  [776] = {x=-522, y=87.731, z=176, rx=180, rz=-85.738, shoulder=lefty, elbow=epositive, wrist=wpositive, fatherId=fReference[0]}
  [777] = {x=-519.753, y=117.878, z=176, rx=180, rz=-72.47, shoulder=lefty, elbow=epositive, wrist=wpositive, fatherId=fReference[0]}
  [778] = {x=-510.651, y=146.693, z=176, rx=180, rz=-58.912, shoulder=lefty, elbow=epositive, wrist=wpositive, fatherId=fReference[0]}
  [779] = {x=-495.048, y=172.571, z=176, rx=180, rz=-45.354, shoulder=lefty, elbow=epositive, wrist=wpositive, fatherId=fReference[0]}
  [780] = {x=-473.813, y=194.069, z=176, rx=180, rz=-31.796, shoulder=lefty, elbow=epositive, wrist=wpositive, fatherId=fReference[0]}
  [781] = {x=-448.13, y=209.991, z=176, rx=180, rz=-18.238, shoulder=lefty, elbow=epositive, wrist=wpositive, fatherId=fReference[0]}
  [782] = {x=-419.43, y=219.448, z=176, rx=180, rz=-4.843, shoulder=lefty, elbow=epositive, wrist=wpositive, fatherId=fReference[0]}
  [783] = {x=-389.312, y=222, z=176, rx=180, shoulder=lefty, elbow=epositive, wrist=wpositive, fatherId=fReference[0]}
  [784] = {x=-359.024, y=222, z=176, rx=180, shoulder=lefty, elbow=epositive, wrist=wpositive, fatherId=fReference[0]}
  [785] = {x=-328.735, y=222, z=176, rx=-180, shoulder=lefty, elbow=epositive, wrist=wpositive, fatherId=fReference[0]}
  [786] = {x=-298.447, y=222, z=176, rx=180, shoulder=lefty, elbow=epositive, wrist=wpositive, fatherId=fReference[0]}
  [787] = {x=-268.159, y=222, z=176, rx=180, shoulder=lefty, elbow=epositive, wrist=wpositive, fatherId=fReference[0]}
  [788] = {x=-237.87, y=222, z=176, rx=-180, shoulder=lefty, elbow=epositive, wrist=wpositive, fatherId=fReference[0]}
  [789] = {x=-207.582, y=222, z=176, rx=180, shoulder=lefty, elbow=epositive, wrist=wpositive, fatherId=fReference[0]}
  [790] = {x=-177.293, y=222, z=176, rx=180, shoulder=lefty, elbow=epositive, wrist=wpositive, fatherId=fReference[0]}
  [791] = {x=-147.005, y=222, z=176, rx=-180, shoulder=lefty, elbow=epositive, wrist=wpositive, fatherId=fReference[0]}
  [792] = {x=-116.716, y=222, z=176, rx=180, shoulder=lefty, elbow=epositive, wrist=wpositive, fatherId=fReference[0]}
  [793] = {x=-86.428, y=222, z=176, rx=180, shoulder=lefty, elbow=epositive, wrist=wpositive, fatherId=fReference[0]}
  [794] = {x=-56.139, y=222, z=176, rx=180, shoulder=lefty, elbow=epositive, wrist=wpositive, fatherId=fReference[0]}
  [795] = {x=-25.851, y=222, z=176, rx=-180, shoulder=lefty, elbow=epositive, wrist=wpositive, fatherId=fReference[0]}
  [796] = {x=4.437, y=222, z=176, rx=-180, shoulder=lefty, elbow=epositive, wrist=wpositive, fatherId=fReference[0]}
  [797] = {x=34.726, y=222, z=176, rx=-180, shoulder=lefty, elbow=epositive, wrist=wpositive, fatherId=fReference[0]}
  [798] = {x=65.014, y=222, z=176, rx=180, shoulder=lefty, elbow=epositive, wrist=wpositive, fatherId=fReference[0]}
  [799] = {x=95.303, y=222, z=176, rx=180, shoulder=lefty, elbow=epositive, wrist=wpositive, fatherId=fReference[0]}
  [800] = {x=125.591, y=222, z=176, rx=-180, shoulder=lefty, elbow=epositive, wrist=wpositive, fatherId=fReference[0]}
  [801] = {x=155.88, y=222, z=176, rx=180, shoulder=lefty, elbow=epositive, wrist=wpositive, fatherId=fReference[0]}
  [802] = {x=186.168, y=222, z=176, rx=180, shoulder=lefty, elbow=epositive, wrist=wpositive, fatherId=fReference[0]}
  [803] = {x=216.456, y=222, z=176, rx=180, shoulder=lefty, elbow=epositive, wrist=wpositive, fatherId=fReference[0]}
  [804] = {x=246.745, y=222, z=176, rx=180, shoulder=lefty, elbow=epositive, wrist=wpositive, fatherId=fReference[0]}
  [805] = {x=277.033, y=222, z=176, rx=180, shoulder=lefty, elbow=epositive, wrist=wpositive, fatherId=fReference[0]}
  [806] = {x=307.322, y=222, z=176, rx=-180, shoulder=lefty, elbow=epositive, wrist=wpositive, fatherId=fReference[0]}
  [807] = {x=337.61, y=222, z=176, rx=180, shoulder=lefty, elbow=epositive, wrist=wpositive, fatherId=fReference[0]}
  [808] = {x=367.899, y=222, z=176, rx=-180, rz=0.13, shoulder=lefty, elbow=epositive, wrist=wpositive, fatherId=fReference[0]}
  [809] = {x=398.186, y=221.932, z=176, rx=180, rz=8.653, shoulder=lefty, elbow=epositive, wrist=wpositive, fatherId=fReference[0]}
  [810] = {x=428.06, y=217.385, z=176, rx=180, rz=22.211, shoulder=lefty, elbow=epositive, wrist=wpositive, fatherId=fReference[0]}
  [811] = {x=456.036, y=205.962, z=176, rx=-180, rz=35.769, shoulder=lefty, elbow=epositive, wrist=wpositive, fatherId=fReference[0]}
  [812] = {x=480.554, y=188.3, z=176, rx=-180, rz=49.327, shoulder=lefty, elbow=epositive, wrist=wpositive, fatherId=fReference[0]}
  [813] = {x=500.248, y=165.381, z=176, rx=180, rz=62.884, shoulder=lefty, elbow=epositive, wrist=wpositive, fatherId=fReference[0]}
  [814] = {x=514.021, y=138.485, z=176, rx=-180, rz=76.442, shoulder=lefty, elbow=epositive, wrist=wpositive, fatherId=fReference[0]}
  [815] = {x=521.105, y=109.109, z=176, rx=-180, rz=88.306, shoulder=lefty, elbow=epositive, wrist=wpositive, fatherId=fReference[0]}
  [816] = {x=522, y=78.856, z=176, rx=180, rz=90, shoulder=lefty, elbow=epositive, wrist=wpositive, fatherId=fReference[0]}
  [817] = {x=522, y=48.567, z=176, rx=180, rz=90, shoulder=lefty, elbow=epositive, wrist=wpositive, fatherId=fReference[0]}
  [818] = {x=522, y=18.279, z=176, rx=180, rz=90, shoulder=lefty, elbow=epositive, wrist=wpositive, fatherId=fReference[0]}
  [819] = {x=522, y=-12.01, z=176, rx=180, rz=90, shoulder=lefty, elbow=epositive, wrist=wpositive, fatherId=fReference[0]}
  [820] = {x=522, y=-42.298, z=176, rx=180, rz=90, shoulder=lefty, elbow=epositive, wrist=wpositive, fatherId=fReference[0]}
  [821] = {x=522, y=-72.586, z=176, rx=180, rz=90.582, shoulder=lefty, elbow=epositive, wrist=wpositive, fatherId=fReference[0]}
  [822] = {x=521.692, y=-102.868, z=176, rx=180, rz=100.751, shoulder=lefty, elbow=epositive, wrist=wpositive, fatherId=fReference[0]}
  [823] = {x=516.055, y=-132.555, z=176, rx=180, rz=114.309, shoulder=lefty, elbow=epositive, wrist=wpositive, fatherId=fReference[0]}
  [824] = {x=503.616, y=-160.094, z=176, rx=180, rz=127.867, shoulder=lefty, elbow=epositive, wrist=wpositive, fatherId=fReference[0]}
  [825] = {x=485.067, y=-183.949, z=176, rx=180, rz=141.425, shoulder=lefty, elbow=epositive, wrist=wpositive, fatherId=fReference[0]}
  [826] = {x=461.443, y=-202.791, z=176, rx=180, rz=154.983, shoulder=lefty, elbow=epositive, wrist=wpositive, fatherId=fReference[0]}
  [827] = {x=434.06, y=-215.57, z=176, rx=-180, rz=168.541, shoulder=lefty, elbow=epositive, wrist=wpositive, fatherId=fReference[0]}
  [828] = {x=404.445, y=-221.573, z=176, rx=-180, rz=176.192, shoulder=lefty, elbow=epositive, wrist=wpositive, fatherId=fReference[0]}
  [829] = {x=374.168, y=-222, z=176, rx=-180, rz=177, shoulder=lefty, elbow=epositive, wrist=wpositive, fatherId=fReference[0]}
  [830] = {x=343.88, y=-222, z=176, rx=-180, rz=178, shoulder=lefty, elbow=epositive, wrist=wpositive, fatherId=fReference[0]}
  [831] = {x=313.591, y=-222, z=176, rx=-180, rz=179, shoulder=lefty, elbow=epositive, wrist=wpositive, fatherId=fReference[0]}
  [832] = {x=283.303, y=-222, z=176, rx=180, rz=-180, shoulder=lefty, elbow=epositive, wrist=wpositive, fatherId=fReference[0]}
  [833] = {x=253.014, y=-222, z=176, rx=180, rz=-180, shoulder=lefty, elbow=epositive, wrist=wpositive, fatherId=fReference[0]}
  [834] = {x=222.726, y=-222, z=176, rx=-180, rz=-180, shoulder=lefty, elbow=epositive, wrist=wpositive, fatherId=fReference[0]}
  [835] = {x=192.437, y=-222, z=176, rx=-180, rz=-180, shoulder=lefty, elbow=epositive, wrist=wpositive, fatherId=fReference[0]}
  [836] = {x=162.149, y=-222, z=176, rx=180, rz=-180, shoulder=lefty, elbow=epositive, wrist=wpositive, fatherId=fReference[0]}
  [837] = {x=131.861, y=-222, z=176, rx=-180, rz=-180, shoulder=lefty, elbow=epositive, wrist=wpositive, fatherId=fReference[0]}
  [838] = {x=101.572, y=-222, z=176, rx=180, rz=-180, shoulder=lefty, elbow=epositive, wrist=wpositive, fatherId=fReference[0]}
  [839] = {x=71.284, y=-222, z=176, rx=-180, rz=-180, shoulder=lefty, elbow=epositive, wrist=wpositive, fatherId=fReference[0]}
  [840] = {x=40.995, y=-222, z=176, rx=180, rz=-180, shoulder=lefty, elbow=epositive, wrist=wpositive, fatherId=fReference[0]}
  [841] = {x=10.707, y=-222, z=176, rx=180, rz=-180, shoulder=lefty, elbow=epositive, wrist=wpositive, fatherId=fReference[0]}
  [842] = {x=-19.582, y=-222, z=176, rx=180, rz=-180, shoulder=lefty, elbow=epositive, wrist=wpositive, fatherId=fReference[0]}
  [843] = {x=-49.87, y=-222, z=176, rx=-180, rz=-180, shoulder=lefty, elbow=epositive, wrist=wpositive, fatherId=fReference[0]}
  [844] = {x=-80.159, y=-222, z=176, rx=-180, rz=-180, shoulder=lefty, elbow=epositive, wrist=wpositive, fatherId=fReference[0]}
  [845] = {x=-110.447, y=-222, z=176, rx=180, rz=-180, shoulder=lefty, elbow=epositive, wrist=wpositive, fatherId=fReference[0]}
  [846] = {x=-140.735, y=-222, z=176, rx=180, rz=-180, shoulder=lefty, elbow=epositive, wrist=wpositive, fatherId=fReference[0]}
  [847] = {x=-171.024, y=-222, z=176, rx=180, rz=-180, shoulder=lefty, elbow=epositive, wrist=wpositive, fatherId=fReference[0]}
  [848] = {x=-201.312, y=-222, z=176, rx=180, rz=-180, shoulder=lefty, elbow=epositive, wrist=wpositive, fatherId=fReference[0]}
  [849] = {x=-231.601, y=-222, z=176, rx=180, rz=-180, shoulder=lefty, elbow=epositive, wrist=wpositive, fatherId=fReference[0]}
  [850] = {x=-261.889, y=-222, z=176, rx=-180, rz=-180, shoulder=lefty, elbow=epositive, wrist=wpositive, fatherId=fReference[0]}
  [851] = {x=-292.178, y=-222, z=176, rx=180, rz=-180, shoulder=lefty, elbow=epositive, wrist=wpositive, fatherId=fReference[0]}
  [852] = {x=-322.466, y=-222, z=176, rx=180, rz=-180, shoulder=lefty, elbow=epositive, wrist=wpositive, fatherId=fReference[0]}
  [853] = {x=-352.754, y=-222, z=176, rx=-180, rz=-180, shoulder=lefty, elbow=epositive, wrist=wpositive, fatherId=fReference[0]}
  [854] = {x=-383.043, y=-222, z=176, rx=-180, rz=-177.239, shoulder=lefty, elbow=epositive, wrist=wpositive, fatherId=fReference[0]}
  [855] = {x=-413.258, y=-220.543, z=176, rx=180, rz=-164.568, shoulder=lefty, elbow=epositive, wrist=wpositive, fatherId=fReference[0]}
  [856] = {x=-442.386, y=-212.502, z=176, rx=180, rz=-157.01, shoulder=lefty, elbow=epositive, wrist=wpositive, fatherId=fReference[0]}
  [857] = {x=-468.818, y=-197.857, z=176, rx=-180, rz=-156.452, shoulder=lefty, elbow=epositive, wrist=wpositive, fatherId=fReference[0]}
  [858] = {x=-491.08, y=-177.424, z=176, rx=180, rz=-154.895, shoulder=lefty, elbow=epositive, wrist=wpositive, fatherId=fReference[0]}
  [859] = {x=-507.931, y=-152.341, z=176, rx=-180, rz=-154.337, shoulder=lefty, elbow=epositive, wrist=wpositive, fatherId=fReference[0]}
  [860] = {x=-518.433, y=-124.007, z=176, rx=180, rz=-153.779, shoulder=lefty, elbow=epositive, wrist=wpositive, fatherId=fReference[0]}
  [861] = {x=-522, y=-94, z=176, rx=180, rz=-152.779, shoulder=lefty, elbow=epositive, wrist=wpositive, fatherId=fReference[0]}
  [862] = {x=-522, y=-94, z=176, rx=180, rz=-152.779, shoulder=lefty, elbow=epositive, wrist=wpositive, fatherId=fReference[0]}
  [863] = {x=-522, y=-94, z=276, rx=-180, rz=-152.779, shoulder=lefty, elbow=epositive, wrist=wpositive, fatherId=fReference[0]}
  [864] = {x=-477.591, y=-88.721, z=287.443, rx=176.622, ry=-26.365, rz=160.43, shoulder=lefty, elbow=epositive, wrist=wpositive, fatherId=fReference[0]}
  [865] = {x=-522, y=-94, z=198, rx=176.622, ry=-26.365, rz=-18.57, shoulder=lefty, elbow=epositive, wrist=wpositive, fatherId=fReference[0]}
  [866] = {x=-522, y=-94, z=198, rx=176.622, ry=-26.365, rz=-97.57, shoulder=lefty, elbow=epositive, wrist=wpositive, fatherId=fReference[0]}
  [867] = {x=-518.433, y=-124.007, z=198, rx=176.622, ry=-26.365, rz=-109.742, shoulder=lefty, elbow=epositive, wrist=wpositive, fatherId=fReference[0]}
  [868] = {x=-507.931, y=-152.341, z=198, rx=170.142, ry=-24.793, rz=-124.68, shoulder=lefty, elbow=epositive, wrist=wpositive, fatherId=fReference[0]}
  [869] = {x=-491.08, y=-177.424, z=198, rx=164.42, ry=-21.791, rz=-139.083, shoulder=lefty, elbow=epositive, wrist=wpositive, fatherId=fReference[0]}
  [870] = {x=-468.818, y=-197.857, z=198, rx=159.778, ry=-17.602, rz=-152.787, shoulder=lefty, elbow=epositive, wrist=wpositive, fatherId=fReference[0]}
  [871] = {x=-442.386, y=-212.502, z=198, rx=156.378, ry=-12.518, rz=-165.809, shoulder=lefty, elbow=epositive, wrist=wpositive, fatherId=fReference[0]}
  [872] = {x=-413.258, y=-220.543, z=198, rx=154.267, ry=-6.834, rz=-177.501, shoulder=lefty, elbow=epositive, wrist=wpositive, fatherId=fReference[0]}
  [873] = {x=-383.043, y=-222, z=198, rx=153.462, ry=-1.234, rz=-180, shoulder=lefty, elbow=epositive, wrist=wpositive, fatherId=fReference[0]}
  [874] = {x=-352.754, y=-222, z=198, rx=153.435, rz=-180, shoulder=lefty, elbow=epositive, wrist=wpositive, fatherId=fReference[0]}
  [875] = {x=-322.466, y=-222, z=198, rx=153.435, rz=-180, shoulder=lefty, elbow=epositive, wrist=wpositive, fatherId=fReference[0]}
  [876] = {x=-292.178, y=-222, z=198, rx=153.435, rz=-180, shoulder=lefty, elbow=epositive, wrist=wpositive, fatherId=fReference[0]}
  [877] = {x=-261.889, y=-222, z=198, rx=153.435, rz=-180, shoulder=lefty, elbow=epositive, wrist=wpositive, fatherId=fReference[0]}
  [878] = {x=-231.601, y=-222, z=198, rx=153.435, rz=-180, shoulder=lefty, elbow=epositive, wrist=wpositive, fatherId=fReference[0]}
  [879] = {x=-201.312, y=-222, z=198, rx=153.435, rz=-180, shoulder=lefty, elbow=epositive, wrist=wpositive, fatherId=fReference[0]}
  [880] = {x=-171.024, y=-222, z=198, rx=153.435, rz=-180, shoulder=lefty, elbow=epositive, wrist=wpositive, fatherId=fReference[0]}
  [881] = {x=-140.735, y=-222, z=198, rx=153.435, rz=-180, shoulder=lefty, elbow=epositive, wrist=wpositive, fatherId=fReference[0]}
  [882] = {x=-110.447, y=-222, z=198, rx=153.435, rz=-180, shoulder=lefty, elbow=epositive, wrist=wpositive, fatherId=fReference[0]}
  [883] = {x=-80.159, y=-222, z=198, rx=153.435, rz=-180, shoulder=lefty, elbow=epositive, wrist=wpositive, fatherId=fReference[0]}
  [884] = {x=-49.87, y=-222, z=198, rx=153.435, rz=-180, shoulder=lefty, elbow=epositive, wrist=wpositive, fatherId=fReference[0]}
  [885] = {x=-19.582, y=-222, z=198, rx=153.435, rz=-180, shoulder=lefty, elbow=epositive, wrist=wpositive, fatherId=fReference[0]}
  [886] = {x=10.707, y=-222, z=198, rx=153.435, rz=-180, shoulder=lefty, elbow=epositive, wrist=wpositive, fatherId=fReference[0]}
  [887] = {x=40.995, y=-222, z=198, rx=153.435, rz=-180, shoulder=lefty, elbow=epositive, wrist=wpositive, fatherId=fReference[0]}
  [888] = {x=71.284, y=-222, z=198, rx=153.435, rz=-180, shoulder=lefty, elbow=epositive, wrist=wpositive, fatherId=fReference[0]}
  [889] = {x=101.572, y=-222, z=198, rx=153.435, rz=-180, shoulder=lefty, elbow=epositive, wrist=wpositive, fatherId=fReference[0]}
  [890] = {x=131.861, y=-222, z=198, rx=153.435, rz=-180, shoulder=lefty, elbow=epositive, wrist=wpositive, fatherId=fReference[0]}
  [891] = {x=162.149, y=-222, z=198, rx=153.435, rz=-180, shoulder=lefty, elbow=epositive, wrist=wpositive, fatherId=fReference[0]}
  [892] = {x=192.437, y=-222, z=198, rx=153.435, rz=-180, shoulder=lefty, elbow=epositive, wrist=wpositive, fatherId=fReference[0]}
  [893] = {x=222.726, y=-222, z=198, rx=153.435, rz=-180, shoulder=lefty, elbow=epositive, wrist=wpositive, fatherId=fReference[0]}
  [894] = {x=253.014, y=-222, z=198, rx=153.435, rz=-180, shoulder=lefty, elbow=epositive, wrist=wpositive, fatherId=fReference[0]}
  [895] = {x=283.303, y=-222, z=198, rx=153.435, rz=-180, shoulder=lefty, elbow=epositive, wrist=wpositive, fatherId=fReference[0]}
  [896] = {x=313.591, y=-222, z=198, rx=153.435, rz=-175, shoulder=lefty, elbow=epositive, wrist=wpositive, fatherId=fReference[0]}
  [897] = {x=343.88, y=-222, z=198, rx=153.435, rz=-166, shoulder=lefty, elbow=epositive, wrist=wpositive, fatherId=fReference[0]}
  [898] = {x=374.168, y=-222, z=198, rx=153.435, rz=-157.722, shoulder=lefty, elbow=epositive, wrist=wpositive, fatherId=fReference[0]}
  [899] = {x=404.445, y=-221.573, z=198, rx=153.437, ry=0.361, rz=-156.272, shoulder=lefty, elbow=epositive, wrist=wpositive, fatherId=fReference[0]}
  [900] = {x=434.06, y=-215.57, z=198, rx=153.894, ry=5.097, rz=157.552, shoulder=lefty, elbow=epositive, wrist=wpositive, fatherId=fReference[0]}
  [901] = {x=461.443, y=-202.791, z=198, rx=155.625, ry=10.902, rz=145.173, shoulder=lefty, elbow=epositive, wrist=wpositive, fatherId=fReference[0]}
  [902] = {x=485.067, y=-183.949, z=198, rx=158.65, ry=16.192, rz=132.325, shoulder=lefty, elbow=epositive, wrist=wpositive, fatherId=fReference[0]}
  [903] = {x=503.616, y=-160.094, z=198, rx=162.938, ry=20.674, rz=118.83, shoulder=lefty, elbow=epositive, wrist=wpositive, fatherId=fReference[0]}
  [904] = {x=516.055, y=-132.555, z=198, rx=168.369, ry=24.052, rz=104.624, shoulder=lefty, elbow=epositive, wrist=wpositive, fatherId=fReference[0]}
  [905] = {x=521.692, y=-102.868, z=198, rx=174.671, ry=26.063, rz=92.871, shoulder=lefty, elbow=epositive, wrist=wpositive, fatherId=fReference[0]}
  [906] = {x=522, y=-72.586, z=198, rx=179.709, ry=26.564, rz=90.13, shoulder=lefty, elbow=epositive, wrist=wpositive, fatherId=fReference[0]}
  [907] = {x=522, y=-42.298, z=198, rx=180, ry=26.565, rz=90, shoulder=lefty, elbow=epositive, wrist=wpositive, fatherId=fReference[0]}
  [908] = {x=522, y=-12.01, z=198, rx=180, ry=26.565, rz=90, shoulder=lefty, elbow=epositive, wrist=wpositive, fatherId=fReference[0]}
  [909] = {x=522, y=18.279, z=198, rx=180, ry=26.565, rz=90, shoulder=lefty, elbow=epositive, wrist=wpositive, fatherId=fReference[0]}
  [910] = {x=522, y=48.567, z=198, rx=180, ry=26.565, rz=90, shoulder=lefty, elbow=epositive, wrist=wpositive, fatherId=fReference[0]}
  [911] = {x=522, y=78.856, z=198, rx=-180, ry=26.565, rz=88.485, shoulder=lefty, elbow=epositive, wrist=wpositive, fatherId=fReference[0]}
  [912] = {x=521.105, y=109.109, z=198, rx=-179.153, ry=26.553, rz=77.465, shoulder=lefty, elbow=epositive, wrist=wpositive, fatherId=fReference[0]}
  [913] = {x=514.021, y=138.485, z=198, rx=-173.315, ry=25.769, rz=62.74, shoulder=lefty, elbow=epositive, wrist=wpositive, fatherId=fReference[0]}
  [914] = {x=500.248, y=165.381, z=198, rx=-167.162, ry=23.457, rz=48.037, shoulder=lefty, elbow=epositive, wrist=wpositive, fatherId=fReference[0]}
  [915] = {x=480.554, y=188.3, z=198, rx=-161.951, ry=19.827, rz=33.975, shoulder=lefty, elbow=epositive, wrist=wpositive, fatherId=fReference[0]}
  [916] = {x=456.036, y=205.962, z=198, rx=-157.918, ry=15.153, rz=20.624, shoulder=lefty, elbow=epositive, wrist=wpositive, fatherId=fReference[0]}
  [917] = {x=428.06, y=217.385, z=198, rx=-155.161, ry=9.733, rz=7.891, shoulder=lefty, elbow=epositive, wrist=wpositive, fatherId=fReference[0]}
  [918] = {x=398.186, y=221.932, z=198, rx=-153.696, ry=3.858, rz=1.116, shoulder=lefty, elbow=epositive, wrist=wpositive, fatherId=fReference[0]}
  [919] = {x=367.899, y=222, z=198, rx=-153.435, ry=0.058, shoulder=lefty, elbow=epositive, wrist=wpositive, fatherId=fReference[0]}
  [920] = {x=337.61, y=222, z=198, rx=-153.435, shoulder=lefty, elbow=epositive, wrist=wpositive, fatherId=fReference[0]}
  [921] = {x=307.322, y=222, z=198, rx=-153.435, shoulder=lefty, elbow=epositive, wrist=wpositive, fatherId=fReference[0]}
  [922] = {x=277.033, y=222, z=198, rx=-153.435, rz=1, shoulder=lefty, elbow=epositive, wrist=wpositive, fatherId=fReference[0]}
  [923] = {x=246.745, y=222, z=198, rx=-153.435, rz=2, shoulder=lefty, elbow=epositive, wrist=wpositive, fatherId=fReference[0]}
  [924] = {x=216.456, y=222, z=198, rx=-153.435, rz=2, shoulder=lefty, elbow=epositive, wrist=wpositive, fatherId=fReference[0]}
  [925] = {x=186.168, y=222, z=198, rx=-153.435, rz=3, shoulder=lefty, elbow=epositive, wrist=wpositive, fatherId=fReference[0]}
  [926] = {x=155.88, y=222, z=198, rx=-153.435, rz=4, shoulder=lefty, elbow=epositive, wrist=wpositive, fatherId=fReference[0]}
  [927] = {x=125.591, y=222, z=198, rx=-153.435, rz=4, shoulder=lefty, elbow=epositive, wrist=wpositive, fatherId=fReference[0]}
  [928] = {x=95.303, y=222, z=198, rx=-153.435, rz=5, shoulder=lefty, elbow=epositive, wrist=wpositive, fatherId=fReference[0]}
  [929] = {x=65.014, y=222, z=198, rx=-153.435, rz=6, shoulder=lefty, elbow=epositive, wrist=wpositive, fatherId=fReference[0]}
  [930] = {x=34.726, y=222, z=198, rx=-153.435, rz=7, shoulder=lefty, elbow=epositive, wrist=wpositive, fatherId=fReference[0]}
  [931] = {x=4.437, y=222, z=198, rx=-153.435, rz=7, shoulder=lefty, elbow=epositive, wrist=wpositive, fatherId=fReference[0]}
  [932] = {x=-25.851, y=222, z=198, rx=-153.435, rz=8, shoulder=lefty, elbow=epositive, wrist=wpositive, fatherId=fReference[0]}
  [933] = {x=-56.139, y=222, z=198, rx=-153.435, rz=9, shoulder=lefty, elbow=epositive, wrist=wpositive, fatherId=fReference[0]}
  [934] = {x=-86.428, y=222, z=198, rx=-153.435, rz=10, shoulder=lefty, elbow=epositive, wrist=wpositive, fatherId=fReference[0]}
  [935] = {x=-116.716, y=222, z=198, rx=-153.435, rz=10, shoulder=lefty, elbow=epositive, wrist=wpositive, fatherId=fReference[0]}
  [936] = {x=-147.005, y=222, z=198, rx=-153.435, rz=11, shoulder=lefty, elbow=epositive, wrist=wpositive, fatherId=fReference[0]}
  [937] = {x=-177.293, y=222, z=198, rx=-153.435, rz=12, shoulder=lefty, elbow=epositive, wrist=wpositive, fatherId=fReference[0]}
  [938] = {x=-207.582, y=222, z=198, rx=-153.435, rz=13, shoulder=lefty, elbow=epositive, wrist=wpositive, fatherId=fReference[0]}
  [939] = {x=-237.87, y=222, z=198, rx=-153.435, rz=13, shoulder=lefty, elbow=epositive, wrist=wpositive, fatherId=fReference[0]}
  [940] = {x=-268.159, y=222, z=198, rx=-153.435, rz=14, shoulder=lefty, elbow=epositive, wrist=wpositive, fatherId=fReference[0]}
  [941] = {x=-298.447, y=222, z=198, rx=-153.435, rz=15, shoulder=lefty, elbow=epositive, wrist=wpositive, fatherId=fReference[0]}
  [942] = {x=-328.735, y=222, z=198, rx=-153.435, rz=16, shoulder=lefty, elbow=epositive, wrist=wpositive, fatherId=fReference[0]}
  [943] = {x=-359.024, y=222, z=198, rx=-153.435, rz=17, shoulder=lefty, elbow=epositive, wrist=wpositive, fatherId=fReference[0]}
  [944] = {x=-389.312, y=222, z=198, rx=-153.435, rz=17.667, shoulder=lefty, elbow=epositive, wrist=wpositive, fatherId=fReference[0]}
  [945] = {x=-419.43, y=219.448, z=198, rx=-153.517, ry=-2.164, rz=16.642, shoulder=lefty, elbow=epositive, wrist=wpositive, fatherId=fReference[0]}
  [946] = {x=-448.13, y=209.991, z=198, rx=-154.598, ry=-8.046, rz=13.406, shoulder=lefty, elbow=epositive, wrist=wpositive, fatherId=fReference[0]}
  [947] = {x=-473.813, y=194.069, z=198, rx=-156.976, ry=-13.629, rz=8.821, shoulder=lefty, elbow=epositive, wrist=wpositive, fatherId=fReference[0]}
  [948] = {x=-495.048, y=172.571, z=198, rx=-160.64, ry=-18.553, rz=2.666, shoulder=lefty, elbow=epositive, wrist=wpositive, fatherId=fReference[0]}
  [949] = {x=-510.651, y=146.693, z=198, rx=-165.524, ry=-22.519, rz=-5.186, shoulder=lefty, elbow=epositive, wrist=wpositive, fatherId=fReference[0]}
  [950] = {x=-519.753, y=117.878, z=198, rx=-171.435, ry=-25.242, rz=-13.458, shoulder=lefty, elbow=epositive, wrist=wpositive, fatherId=fReference[0]}
  [951] = {x=-522, y=87.731, z=198, rx=-177.872, ry=-26.486, rz=-24.05, shoulder=lefty, elbow=epositive, wrist=wpositive, fatherId=fReference[0]}
  [952] = {x=-522, y=57.442, z=198, rx=-180, ry=-26.565, rz=-26, shoulder=lefty, elbow=epositive, wrist=wpositive, fatherId=fReference[0]}
  [953] = {x=-522, y=27.154, z=198, rx=180, ry=-26.565, rz=-23, shoulder=lefty, elbow=epositive, wrist=wpositive, fatherId=fReference[0]}
  [954] = {x=-522, y=-3.135, z=198, rx=180, ry=-26.565, rz=-21, shoulder=lefty, elbow=epositive, wrist=wpositive, fatherId=fReference[0]}
  [955] = {x=-522, y=-33.423, z=198, rx=180, ry=-26.565, rz=-18, shoulder=lefty, elbow=epositive, wrist=wpositive, fatherId=fReference[0]}
  [956] = {x=-522, y=-63.712, z=198, rx=180, ry=-26.565, rz=-16, shoulder=lefty, elbow=epositive, wrist=wpositive, fatherId=fReference[0]}
  [957] = {x=-522, y=-94, z=198, rx=180, ry=-26.565, rz=-14, shoulder=lefty, elbow=epositive, wrist=wpositive, fatherId=fReference[0]}
  [958] = {x=-522, y=-94, z=198, rx=180, ry=-26.565, rz=-14, shoulder=lefty, elbow=epositive, wrist=wpositive, fatherId=fReference[0]}
  [959] = {x=-477.279, y=-94, z=287.443, rx=180, ry=-26.565, rz=-14, shoulder=lefty, elbow=epositive, wrist=wpositive, fatherId=fReference[0]}
public tool tTool = {z=452, fatherId=flange[0], ioLink=valve1}
aio Tpompe = {link=CanIO\RemIO\remio0_QW}
aio Tpompe1 = {link=CanIO\RemIO\remio0_QW}
aio Tpompe2 = {link=CanIO\RemIO\remio0_QW}
aio Tpompe3 = {link=CanIO\RemIO\remio0_QW}
aio Tpompe4 = {link=CanIO\RemIO\remio0_QW}
aio Tpompe5 = {link=CanIO\RemIO\remio0_QW}
dio doPompe = {link=CanIO\RemIO\remio0_Q}
dio doPompe1 = {link=CanIO\RemIO\remio0_Q}
dio doValve1 = {link=valve1}
dio doValve2 = {link=valve2}
aio Tpompe6 = {link=CanIO\RemIO\remio0_QW}
aio Tpompe7 = {link=CanIO\RemIO\remio0_QW}
aio Tpompe8 = {link=CanIO\RemIO\remio0_QW}
dio doPompe2 = {link=CanIO\RemIO\remio0_Q}
dio doPompe3 = {link=CanIO\RemIO\remio0_Q}
dio doValve3 = {link=valve1}
dio doValve4 = {link=valve2}
num nTension = 1.2
num nTObtOpen = 2
num nTPompeOff = 2
num nTPompeOn = 2
